PROGRAM GameEngine
VAR
	fbSnake			: FB_Snake;
	fbFood			: FB_Food;
	fbDraw			: FB_Draw;
	
	updateTimer		: TON;
	bSnakeMove		: BOOL;

	rTrig			: R_TRIG;
END_VAR

rTrig(CLK := GVL_Variables.bInit);
fbSnake(aStSnakeBody:= GVL_Variables.aStSnakeBody, iSnakeLength := GVL_Variables.iSnakeLength);
fbFood(stFood => GVL_Variables.stFood);

IF rTrig.Q THEN
	GVL_Variables.aStSnakeBody := GVL_Variables.aStSnakeBodyEmpty;
	GVL_Variables.aStSnakeBody[1].stBodyCoordinate.iColumnCoordinate := 5;
	GVL_Variables.aStSnakeBody[1].stBodyCoordinate.iRowCoordinate := 5;
	GVL_Variables.iSnakeLength := 1;
	GVL_Variables.bGameOver := FALSE;
	GVL_Variables.bInit := FALSE;
END_IF

IF NOT GVL_Variables.bGameOver THEN
	updateTimer(IN := NOT updateTimer.Q, PT := T#1S);
	IF updateTimer.Q THEN
		bSnakeMove := fbSnake.M_Move(GVL_Variables.iSnakeDirection);		
	END_IF

	IF fbSnake.M_Die() THEN
		GVL_Variables.bGameOver := TRUE;
	END_IF

	IF fbSnake.M_Eat(GVL_Variables.stFood) THEN
		fbFood.M_Generate();
	END_IF
END_IF

fbDraw();
GVL_Variables.bDraw := fbDraw.M_Draw();

END_PROGRAM

(* stored: Version 1.1.0.1, ProductVersion 3.1.4024.4
   POU GameEngine: Id {f3d1851b-2b90-41cf-9e90-238148830b16}, SpecialFunc None *)
